TYPE AdasConfiguration :
STRUCT
	track: ARRAY[0..(gVarL.gVar_NumberOfAdasTracks - 1)] OF BYTE;
	signal: ARRAY[0..(gVarL.gVar_NumberOfAdasTracks - 1)] OF BYTE;
	axis: ARRAY[0..(gVarL.gVar_NumberOfAdasTracks - 1)] OF BYTE;
END_STRUCT
END_TYPE

(* stored: Version 1.1.0.1, ProductVersion 3.1.4022.16
   DUT AdasConfiguration: Id {35369538-4177-4379-988d-99c8d13282ab} *)
